GLOBALCONSTANTS myPorts_espnow (* Global constants *)
  (* Standard: 61499-1; Description: Copyright (c) 2023 HR Agrartechnik GmbH This program and the accompanying materials are made available under the terms of the Eclipse Public License 2.0 which is available at https://www.eclipse.org/legal/epl-2.0/ SPDX-License-Identifier: EPL-2.0 *)
  (* Version 1.0, 2023-10-22, Franz Höpfinger, HR Agrartechnik GmbH *)
  PACKAGE VV::const::ports;
  VAR_GLOBAL CONSTANT
    PORT_0_espnow : WSTRING := "fbdk[].espnow[239.0.0.1:61000]";
    PORT_1_espnow : WSTRING := "fbdk[].espnow[239.0.0.1:61001]";
    PORT_2_espnow : WSTRING := "fbdk[].espnow[239.0.0.1:61002]";
    PORT_3_espnow : WSTRING := "fbdk[].espnow[239.0.0.1:61003]";
  END_VAR
END_GLOBALCONSTANTS
